{attribute 'TcGenerated'}
{attribute 'no-analysis'}
{attribute 'linkalways'}
// This function has been automatically generated from the project information.
VAR_GLOBAL CONSTANT
	{attribute 'const_non_replaced'}
	stLibVersion_Servo : ST_LibVersion := (iMajor := 1, iMinor := 0, iBuild := 0, iRevision := 4, nFlags := 1, sVersion := '1.0.0.4');
END_VAR

(* stored: Version 1.1.0.1, ProductVersion 3.1.4024.12
   GVL Global_Version: Id {da3537ae-6446-0de3-1b1e-60f69a2d2f70} *)
